TYPE AxesConfigs_1 :
STRUCT
	IoStageAxisConfig : IoStageAxisConfig;	
	IoDoorSlitAxisConfig : IoDoorSlitAxisConfig;
END_STRUCT
END_TYPE

(* stored: Version 1.1.0.1, ProductVersion 3.1.4024.12
   DUT AxesConfigs_1: Id {1354407f-b781-4182-80e6-2e979a424516} *)
